TYPE stBH0LPL_Line EXTENDS stPIM_LineEventsModule :
STRUCT

	{attribute 'OPC.UA.DA' := '1'}
	stStation_BH0LPL01 : stPIM_StationEventsModule_3_Machine;
END_STRUCT
END_TYPE

(* stored: Version 1.1.0.1, ProductVersion 3.1.4024.15
   DUT stBH0LPL_Line: Id {fc951564-ef85-405c-bf8b-388816988ad2} *)
